{attribute 'qualified_only'}
{attribute 'strict'}
TYPE e_NciChannelError :
(
  e_Null,
  e_InvalidReference_ChannelRef,
  e_AxisConfigurationMismatch_McAxis,
  e_AxisConfigurationMismatch_AuxAxis


);
END_TYPE

(* stored: Version 1.1.0.1, ProductVersion 3.1.4024.9
   DUT e_NciChannelError: Id {2d3dc3c9-5d65-0533-372b-b9628aaf8da6} *)
